// TIA Portal V20 export
DATA_BLOCK "InstInterfaceSignals"   // DB29
{ DB_Accessible_From_OPC_UA := 'FALSE' }
AUTHOR : SICAR
FAMILY : Diag
VERSION : 1.0
// stored: DBAccessibleFromOPCUA false, DBAccessibleFromWebserver false, InstanceOfName CallInterfaceSignals, InstanceOfType FB
"CallInterfaceSignals"
   // VAR
   //    statReadValueHmi : Bool;
   //    statSelectSignalsHmi : USInt;
   //    statSelectSignalsOld { ExternalAccessible := 'False'; ExternalVisible := 'False'; ExternalWritable := 'False'} : USInt;
   //    statRisEdgeReadName { ExternalAccessible := 'False'; ExternalVisible := 'False'; ExternalWritable := 'False'} : Bool;
   //    statPosPulseReadName : Bool;
   //    statInterfaceSignalsHmi : Array[0..100] of "typeInterfaceSignalsHmi";
   //    instSignals1Left { ExternalAccessible := 'False'; ExternalVisible := 'False'; ExternalWritable := 'False'} : "LAF_InterfaceSignalsBool";
   //    instSignals1Right { ExternalAccessible := 'False'; ExternalVisible := 'False'; ExternalWritable := 'False'} : "LAF_InterfaceSignalsBool";
   //    instSignals2Left { ExternalAccessible := 'False'; ExternalVisible := 'False'; ExternalWritable := 'False'} : "LAF_InterfaceSignalsBool";
   //    instSignals2Right { ExternalAccessible := 'False'; ExternalVisible := 'False'; ExternalWritable := 'False'} : "LAF_InterfaceSignalsBool";
   //    instSignals3Left { ExternalAccessible := 'False'; ExternalVisible := 'False'; ExternalWritable := 'False'} : "LAF_InterfaceSignalsBool";
   //    instSignals3Right { ExternalAccessible := 'False'; ExternalVisible := 'False'; ExternalWritable := 'False'} : "LAF_InterfaceSignalsBool";
   //    instSignals4Left { ExternalAccessible := 'False'; ExternalVisible := 'False'; ExternalWritable := 'False'} : "LAF_InterfaceSignalsBool";
   //    instSignals4Right { ExternalAccessible := 'False'; ExternalVisible := 'False'; ExternalWritable := 'False'} : "LAF_InterfaceSignalsBool";
   //    instSignals5Left { ExternalAccessible := 'False'; ExternalVisible := 'False'; ExternalWritable := 'False'} : "LAF_InterfaceSignalsBool";
   //    instSignals5Right { ExternalAccessible := 'False'; ExternalVisible := 'False'; ExternalWritable := 'False'} : "LAF_InterfaceSignalsBool";
   //    instSignals6Left { S7_SetPoint := 'True'} : "LAF_InterfaceSignalsBool";
   //    instSignals6Right { S7_SetPoint := 'True'} : "LAF_InterfaceSignalsBool";
   //    instSignals7Left { S7_SetPoint := 'True'} : "LAF_InterfaceSignalsBool";
   //    instSignals7Right { S7_SetPoint := 'True'} : "LAF_InterfaceSignalsBool";
   //    instSignals8Left { S7_SetPoint := 'True'} : "LAF_InterfaceSignalsBool";
   //    instSignals8Right { S7_SetPoint := 'True'} : "LAF_InterfaceSignalsBool";
   //    instSignals9Left { S7_SetPoint := 'True'} : "LAF_InterfaceSignalsBool";
   //    instSignals9Right { S7_SetPoint := 'True'} : "LAF_InterfaceSignalsBool";
   //    instSignals10Left_ { S7_SetPoint := 'True'} : "LAF_InterfaceSignalsBool";
   //    instSignals10Right { S7_SetPoint := 'True'} : "LAF_InterfaceSignalsBool";
   //    instSignals11Left { S7_SetPoint := 'True'} : "LAF_InterfaceSignalsBool";
   //    instSignals11Right { S7_SetPoint := 'True'} : "LAF_InterfaceSignalsBool";
   //    instSignals12Left { S7_SetPoint := 'True'} : "LAF_InterfaceSignalsBool";
   //    instSignals12Right { S7_SetPoint := 'True'} : "LAF_InterfaceSignalsBool";
   //    instSignals13Left { S7_SetPoint := 'True'} : "LAF_InterfaceSignalsBool";
   //    instSignals13Right { S7_SetPoint := 'True'} : "LAF_InterfaceSignalsBool";
   //    instSignals14Left { S7_SetPoint := 'True'} : "LAF_InterfaceSignalsBool";
   //    instSignals14Right { S7_SetPoint := 'True'} : "LAF_InterfaceSignalsBool";
   //    instSignals15Left { S7_SetPoint := 'True'} : "LAF_InterfaceSignalsBool";
   //    instSignals15Right { S7_SetPoint := 'True'} : "LAF_InterfaceSignalsBool";
   //    instSignals16Left { S7_SetPoint := 'True'} : "LAF_InterfaceSignalsBool";
   //    instSignals16Right { S7_SetPoint := 'True'} : "LAF_InterfaceSignalsBool";
   //    instSignals17Left { S7_SetPoint := 'True'} : "LAF_InterfaceSignalsBool";
   //    instSignals17Right { S7_SetPoint := 'True'} : "LAF_InterfaceSignalsBool";
   //    instSignals18Left { S7_SetPoint := 'True'} : "LAF_InterfaceSignalsBool";
   //    instSignals18Right { S7_SetPoint := 'True'} : "LAF_InterfaceSignalsBool";
   //    instSignals19Left { S7_SetPoint := 'True'} : "LAF_InterfaceSignalsBool";
   //    instSignals19Right { S7_SetPoint := 'True'} : "LAF_InterfaceSignalsBool";
   //    instSignals20Left { S7_SetPoint := 'True'} : "LAF_InterfaceSignalsBool";
   //    instSignals20Right { S7_SetPoint := 'True'} : "LAF_InterfaceSignalsBool";
   //    instSignals21Left { S7_SetPoint := 'True'} : "LAF_InterfaceSignalsBool";
   //    instSignals21Right { S7_SetPoint := 'True'} : "LAF_InterfaceSignalsBool";
   //    instSignals22Left { S7_SetPoint := 'True'} : "LAF_InterfaceSignalsBool";
   //    instSignals22Right { S7_SetPoint := 'True'} : "LAF_InterfaceSignalsBool";
   //    instSignals23Left { S7_SetPoint := 'True'} : "LAF_InterfaceSignalsBool";
   //    instSignals23Right { S7_SetPoint := 'True'} : "LAF_InterfaceSignalsBool";
   //    instSignals24Left { S7_SetPoint := 'True'} : "LAF_InterfaceSignalsBool";
   //    instSignals24Right { S7_SetPoint := 'True'} : "LAF_InterfaceSignalsBool";
   //    instSignals25Left { S7_SetPoint := 'True'} : "LAF_InterfaceSignalsBool";
   //    instSignals25Right { S7_SetPoint := 'True'} : "LAF_InterfaceSignalsBool";
   //    instSignals26Left { S7_SetPoint := 'True'} : "LAF_InterfaceSignalsBool";
   //    instSignals26Right { S7_SetPoint := 'True'} : "LAF_InterfaceSignalsBool";
   //    instSignals27Left { S7_SetPoint := 'True'} : "LAF_InterfaceSignalsBool";
   //    instSignals27Right { S7_SetPoint := 'True'} : "LAF_InterfaceSignalsBool";
   //    instSignals28Left { S7_SetPoint := 'True'} : "LAF_InterfaceSignalsBool";
   //    instSignals28Right { S7_SetPoint := 'True'} : "LAF_InterfaceSignalsBool";
   //    instSignals29Left { S7_SetPoint := 'True'} : "LAF_InterfaceSignalsBool";
   //    instSignals29Right { S7_SetPoint := 'True'} : "LAF_InterfaceSignalsBool";
   //    instSignals30Left { S7_SetPoint := 'True'} : "LAF_InterfaceSignalsBool";
   //    instSignals30Right { S7_SetPoint := 'True'} : "LAF_InterfaceSignalsBool";
   //    instSignals31Left { S7_SetPoint := 'True'} : "LAF_InterfaceSignalsBool";
   //    instSignals31Right { S7_SetPoint := 'True'} : "LAF_InterfaceSignalsBool";
   //    instSignals32Left { S7_SetPoint := 'True'} : "LAF_InterfaceSignalsBool";
   //    instSignals32Right { S7_SetPoint := 'True'} : "LAF_InterfaceSignalsBool";
   //    instSignals33Left { S7_SetPoint := 'True'} : "LAF_InterfaceSignalsBool";
   //    instSignals33Right { S7_SetPoint := 'True'} : "LAF_InterfaceSignalsBool";
   //    instSignals34Left { S7_SetPoint := 'True'} : "LAF_InterfaceSignalsBool";
   //    instSignals34Right { S7_SetPoint := 'True'} : "LAF_InterfaceSignalsBool";
   //    instSignals35Left { S7_SetPoint := 'True'} : "LAF_InterfaceSignalsBool";
   //    instSignals35Right { S7_SetPoint := 'True'} : "LAF_InterfaceSignalsBool";
   //    instSignals36Left { S7_SetPoint := 'True'} : "LAF_InterfaceSignalsBool";
   //    instSignals36Right { S7_SetPoint := 'True'} : "LAF_InterfaceSignalsBool";
   //    instSignals37Left { S7_SetPoint := 'True'} : "LAF_InterfaceSignalsBool";
   //    instSignals37Right { S7_SetPoint := 'True'} : "LAF_InterfaceSignalsBool";
   //    instSignals38Left { S7_SetPoint := 'True'} : "LAF_InterfaceSignalsBool";
   //    instSignals38Right { S7_SetPoint := 'True'} : "LAF_InterfaceSignalsBool";
   //    instSignals39Left { S7_SetPoint := 'True'} : "LAF_InterfaceSignalsBool";
   //    instSignals39Right { S7_SetPoint := 'True'} : "LAF_InterfaceSignalsBool";
   //    instSignals40Left { S7_SetPoint := 'True'} : "LAF_InterfaceSignalsBool";
   //    instSignals40Right { S7_SetPoint := 'True'} : "LAF_InterfaceSignalsBool";
   //    instSignals41Left { S7_SetPoint := 'True'} : "LAF_InterfaceSignalsBool";
   //    instSignals41Right { S7_SetPoint := 'True'} : "LAF_InterfaceSignalsBool";
   //    instSignals42Left { S7_SetPoint := 'True'} : "LAF_InterfaceSignalsBool";
   //    instSignals42Right { S7_SetPoint := 'True'} : "LAF_InterfaceSignalsBool";
   //    instSignals43Left { S7_SetPoint := 'True'} : "LAF_InterfaceSignalsBool";
   //    instSignals43Right { S7_SetPoint := 'True'} : "LAF_InterfaceSignalsBool";
   //    instSignals44Left { S7_SetPoint := 'True'} : "LAF_InterfaceSignalsBool";
   //    instSignals44Right { S7_SetPoint := 'True'} : "LAF_InterfaceSignalsBool";
   //    instSignals45Left { S7_SetPoint := 'True'} : "LAF_InterfaceSignalsBool";
   //    instSignals45Right { S7_SetPoint := 'True'} : "LAF_InterfaceSignalsBool";
   //    instSignals46Left { S7_SetPoint := 'True'} : "LAF_InterfaceSignalsBool";
   //    instSignals46Right { S7_SetPoint := 'True'} : "LAF_InterfaceSignalsBool";
   //    instSignals47Left { S7_SetPoint := 'True'} : "LAF_InterfaceSignalsBool";
   //    instSignals47Right { S7_SetPoint := 'True'} : "LAF_InterfaceSignalsBool";
   //    instSignals48Left { S7_SetPoint := 'True'} : "LAF_InterfaceSignalsBool";
   //    instSignals48Right { S7_SetPoint := 'True'} : "LAF_InterfaceSignalsBool";
   //    instSignals49Left { S7_SetPoint := 'True'} : "LAF_InterfaceSignalsBool";
   //    instSignals49Right { S7_SetPoint := 'True'} : "LAF_InterfaceSignalsBool";
   //    instSignals50Left { S7_SetPoint := 'True'} : "LAF_InterfaceSignalsBool";
   //    instSignals50Right { S7_SetPoint := 'True'} : "LAF_InterfaceSignalsBool";
   //    instSignals51Left { S7_SetPoint := 'True'} : "LAF_InterfaceSignalsBool";
   //    instSignals51Right { S7_SetPoint := 'True'} : "LAF_InterfaceSignalsBool";
   //    instSignals52Left { S7_SetPoint := 'True'} : "LAF_InterfaceSignalsBool";
   //    instSignals52Right { S7_SetPoint := 'True'} : "LAF_InterfaceSignalsBool";
   //    instSignals53Left { S7_SetPoint := 'True'} : "LAF_InterfaceSignalsBool";
   //    instSignals53Right { S7_SetPoint := 'True'} : "LAF_InterfaceSignalsBool";
   //    instSignals54Left { S7_SetPoint := 'True'} : "LAF_InterfaceSignalsBool";
   //    instSignals54Right { S7_SetPoint := 'True'} : "LAF_InterfaceSignalsBool";
   //    instSignals55Left { S7_SetPoint := 'True'} : "LAF_InterfaceSignalsBool";
   //    instSignals55Right { S7_SetPoint := 'True'} : "LAF_InterfaceSignalsBool";
   //    instSignals56Left { S7_SetPoint := 'True'} : "LAF_InterfaceSignalsBool";
   //    instSignals56Right { S7_SetPoint := 'True'} : "LAF_InterfaceSignalsBool";
   //    instSignals57Left { S7_SetPoint := 'True'} : "LAF_InterfaceSignalsBool";
   //    instSignals57Right { S7_SetPoint := 'True'} : "LAF_InterfaceSignalsBool";
   //    instSignals58Left { S7_SetPoint := 'True'} : "LAF_InterfaceSignalsBool";
   //    instSignals58Right { S7_SetPoint := 'True'} : "LAF_InterfaceSignalsBool";
   //    instSignals59Left { S7_SetPoint := 'True'} : "LAF_InterfaceSignalsBool";
   //    instSignals59Right { S7_SetPoint := 'True'} : "LAF_InterfaceSignalsBool";
   //    instSignals60Left { S7_SetPoint := 'True'} : "LAF_InterfaceSignalsBool";
   //    instSignals60Right { S7_SetPoint := 'True'} : "LAF_InterfaceSignalsBool";
   //    instSignals61Left { S7_SetPoint := 'True'} : "LAF_InterfaceSignalsBool";
   //    instSignals61Right { S7_SetPoint := 'True'} : "LAF_InterfaceSignalsBool";
   //    instSignals62Left { S7_SetPoint := 'True'} : "LAF_InterfaceSignalsBool";
   //    instSignals62Right { S7_SetPoint := 'True'} : "LAF_InterfaceSignalsBool";
   //    instSignals63Left { S7_SetPoint := 'True'} : "LAF_InterfaceSignalsBool";
   //    instSignals63Right { S7_SetPoint := 'True'} : "LAF_InterfaceSignalsBool";
   //    instSignals64Left { S7_SetPoint := 'True'} : "LAF_InterfaceSignalsBool";
   //    instSignals64Right { S7_SetPoint := 'True'} : "LAF_InterfaceSignalsBool";
   //    instSignals65Left { S7_SetPoint := 'True'} : "LAF_InterfaceSignalsBool";
   //    instSignals65Right { S7_SetPoint := 'True'} : "LAF_InterfaceSignalsBool";
   //    instSignals66Left { S7_SetPoint := 'True'} : "LAF_InterfaceSignalsBool";
   //    instSignals66Right { S7_SetPoint := 'True'} : "LAF_InterfaceSignalsBool";
   //    instSignals67Left { S7_SetPoint := 'True'} : "LAF_InterfaceSignalsBool";
   //    instSignals67Right { S7_SetPoint := 'True'} : "LAF_InterfaceSignalsBool";
   //    instSignals68Left { S7_SetPoint := 'True'} : "LAF_InterfaceSignalsBool";
   //    instSignals68Right { S7_SetPoint := 'True'} : "LAF_InterfaceSignalsBool";
   //    instSignals69Left { S7_SetPoint := 'True'} : "LAF_InterfaceSignalsBool";
   //    instSignals69Right { S7_SetPoint := 'True'} : "LAF_InterfaceSignalsBool";
   //    instSignals70Left { S7_SetPoint := 'True'} : "LAF_InterfaceSignalsBool";
   //    instSignals70Right { S7_SetPoint := 'True'} : "LAF_InterfaceSignalsBool";
   //    instSignals71Left { S7_SetPoint := 'True'} : "LAF_InterfaceSignalsBool";
   //    instSignals71Right { S7_SetPoint := 'True'} : "LAF_InterfaceSignalsBool";
   //    instSignals72Left { S7_SetPoint := 'True'} : "LAF_InterfaceSignalsBool";
   //    instSignals72Right { S7_SetPoint := 'True'} : "LAF_InterfaceSignalsBool";
   //    instSignals73Left { S7_SetPoint := 'True'} : "LAF_InterfaceSignalsBool";
   //    instSignals73Right { S7_SetPoint := 'True'} : "LAF_InterfaceSignalsBool";
   //    instSignals74Left { S7_SetPoint := 'True'} : "LAF_InterfaceSignalsBool";
   //    instSignals74Right { S7_SetPoint := 'True'} : "LAF_InterfaceSignalsBool";
   //    instSignals75Left { S7_SetPoint := 'True'} : "LAF_InterfaceSignalsBool";
   //    instSignals75Right { S7_SetPoint := 'True'} : "LAF_InterfaceSignalsBool";
   //    instSignals76Left { S7_SetPoint := 'True'} : "LAF_InterfaceSignalsBool";
   //    instSignals76Right { S7_SetPoint := 'True'} : "LAF_InterfaceSignalsBool";
   // END_VAR
BEGIN
END_DATA_BLOCK
